// TIA Portal V17 export
// export: Created 2025-05-22T06:01:52.7537202Z, ExportSetting WithDefaults, DisplayName Totally Integrated Automation Portal, DisplayVersion V17 Update 8, DisplayName TIA Portal Openness, DisplayVersion V17 Update 8, DisplayName TIA Portal Version Control Interface, DisplayVersion V17, DisplayName SINAMICS Startdrive Advanced, DisplayVersion V17 SP2, DisplayName SINAMICS Startdrive G110M, G120, G120C, G120D, G120P, G115D, DisplayVersion V17 SP2, DisplayName SINAMICS Startdrive G130, G150, S120, S150, SINAMICS MV, S210, DisplayVersion V17 SP2, DisplayName STEP 7 Professional, DisplayVersion V17 Update 8, DisplayName SINUMERIK ONE STEP 7 Toolbox, DisplayVersion V17 Update 12, DisplayName SINUMERIK ONE PLC Basic Program Plus, DisplayVersion V17 Update 12, DisplayName SINUMERIK 840D sl STEP 7 Toolbox, DisplayVersion V17 Update 12, DisplayName STEP 7 Safety, DisplayVersion V17 Update 6, DisplayName WinCC Advanced, DisplayVersion V17 Update 8
FUNCTION "UPTL_EETransline" : Void   // FC1055, LAD
TITLE = UPTL_EETransline
{ S7_Optimized_Access := 'FALSE' }
AUTHOR : Transline
FAMILY : UPTL_Transline
VERSION : 17.0
// Example how to call the LTLP_Transline functions EETransline / Beispiel für den Aufruf der Bausteine aus EETransline
// stored: AutoNumber true, IsIECCheckEnabled false, SetENOAutomatically false, UDAEnableTagReadback false
BEGIN

REGION Network 1: EE Transfer
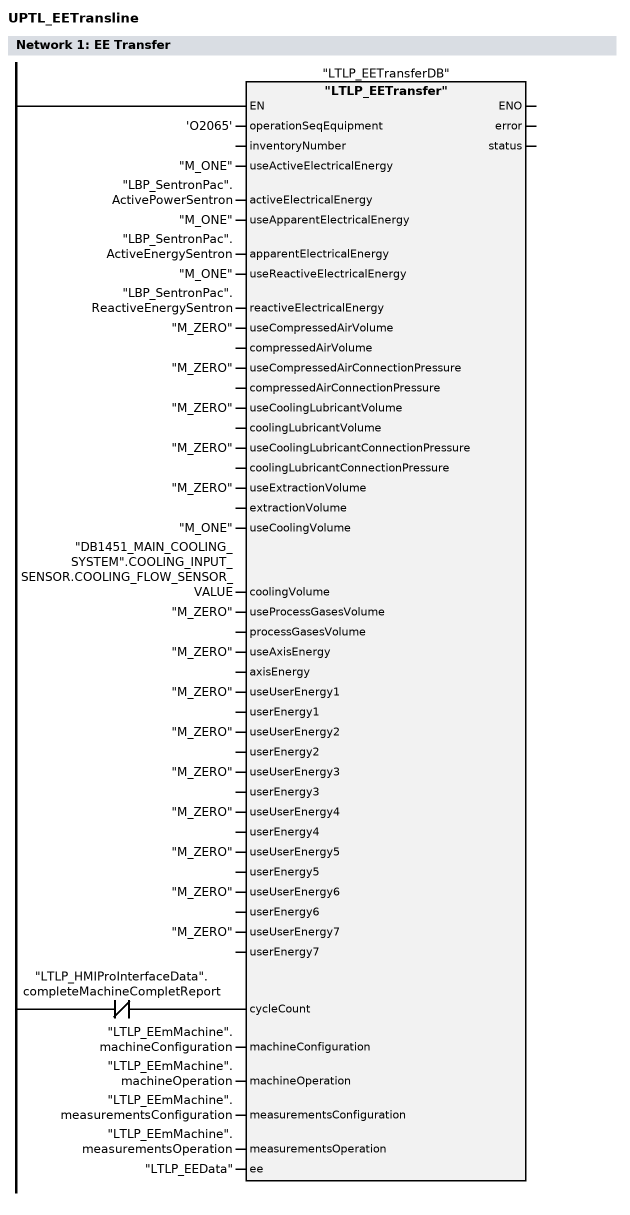
   RUNG wire#powerrail
      "LTLP_EETransferDB"(cycleCount := wire#w1, operationSeqEquipment := 'O2065', inventoryNumber :=, useActiveElectricalEnergy := "M_ONE", activeElectricalEnergy := "LBP_SentronPac".ActivePowerSentron, useApparentElectricalEnergy := "M_ONE", apparentElectricalEnergy := "LBP_SentronPac".ActiveEnergySentron, useReactiveElectricalEnergy := "M_ONE", reactiveElectricalEnergy := "LBP_SentronPac".ReactiveEnergySentron, useCompressedAirVolume := "M_ZERO", compressedAirVolume :=, useCompressedAirConnectionPressure := "M_ZERO", compressedAirConnectionPressure :=, useCoolingLubricantVolume := "M_ZERO", coolingLubricantVolume :=, useCoolingLubricantConnectionPressure := "M_ZERO", coolingLubricantConnectionPressure :=, useExtractionVolume := "M_ZERO", extractionVolume :=, useCoolingVolume := "M_ONE", coolingVolume := "DB1451_MAIN_COOLING_SYSTEM".COOLING_INPUT_SENSOR.COOLING_FLOW_SENSOR_VALUE, useProcessGasesVolume := "M_ZERO", processGasesVolume :=, useAxisEnergy := "M_ZERO", axisEnergy :=, useUserEnergy1 := "M_ZERO", userEnergy1 :=, useUserEnergy2 := "M_ZERO", userEnergy2 :=, useUserEnergy3 := "M_ZERO", userEnergy3 :=, useUserEnergy4 := "M_ZERO", userEnergy4 :=, useUserEnergy5 := "M_ZERO", userEnergy5 :=, useUserEnergy6 := "M_ZERO", userEnergy6 :=, useUserEnergy7 := "M_ZERO", userEnergy7 :=, machineConfiguration := "LTLP_EEmMachine".machineConfiguration, machineOperation := "LTLP_EEmMachine".machineOperation, measurementsConfiguration := "LTLP_EEmMachine".measurementsConfiguration, measurementsOperation := "LTLP_EEmMachine".measurementsOperation, ee := "LTLP_EEData", error =>, status =>)
   END_RUNG
   RUNG wire#powerrail
      I_Contact( "LTLP_HMIProInterfaceData".completeMachineCompletReport )
   END_RUNG wire#w1
   // the same network as SCL:
   "LTLP_EETransferDB"(operationSeqEquipment := 'O2065',   // "LTLP_EETransfer"
                       useActiveElectricalEnergy := "M_ONE",
                       activeElectricalEnergy := "LBP_SentronPac".ActivePowerSentron,
                       useApparentElectricalEnergy := "M_ONE",
                       apparentElectricalEnergy := "LBP_SentronPac".ActiveEnergySentron,
                       useReactiveElectricalEnergy := "M_ONE",
                       reactiveElectricalEnergy := "LBP_SentronPac".ReactiveEnergySentron,
                       useCompressedAirVolume := "M_ZERO",
                       useCompressedAirConnectionPressure := "M_ZERO",
                       useCoolingLubricantVolume := "M_ZERO",
                       useCoolingLubricantConnectionPressure := "M_ZERO",
                       useExtractionVolume := "M_ZERO",
                       useCoolingVolume := "M_ONE",
                       coolingVolume := "DB1451_MAIN_COOLING_SYSTEM".COOLING_INPUT_SENSOR.COOLING_FLOW_SENSOR_VALUE,
                       useProcessGasesVolume := "M_ZERO",
                       useAxisEnergy := "M_ZERO",
                       useUserEnergy1 := "M_ZERO",
                       useUserEnergy2 := "M_ZERO",
                       useUserEnergy3 := "M_ZERO",
                       useUserEnergy4 := "M_ZERO",
                       useUserEnergy5 := "M_ZERO",
                       useUserEnergy6 := "M_ZERO",
                       useUserEnergy7 := "M_ZERO",
                       cycleCount := NOT "LTLP_HMIProInterfaceData".completeMachineCompletReport,
                       machineConfiguration := "LTLP_EEmMachine".machineConfiguration,
                       machineOperation := "LTLP_EEmMachine".machineOperation,
                       measurementsConfiguration := "LTLP_EEmMachine".measurementsConfiguration,
                       measurementsOperation := "LTLP_EEmMachine".measurementsOperation,
                       ee := "LTLP_EEData");
END_REGION
END_FUNCTION
